// Mitsubishi GX Works2 project: 13   PLC: FX3G

// task Task_01 (event TRUE, interval 0, priority 31): POU_01

PROGRAM POU_01
VAR
  wstep : INT;
  ton1 : TON;
  ii : INT;
END_VAR
IF M8002 THEN
	wstep := 0;
END_IF;

IF NOT M0 THEN
	wstep := 0;
END_IF;

CASE wstep OF
	0:
		FOR ii := 0 TO 3 BY 1 DO
			Z0 := ii;
			Y0Z0 := FALSE;
		END_FOR;
		
		IF M0 THEN
			wstep := 20;
		END_IF;
				
	20:
		Y3 := FALSE;
		Y0 := TRUE;
		ton1(IN := TRUE, PT := T#2s);
		IF ton1.Q THEN
			ton1(IN := FALSE);
			wstep := 21;
		END_IF;
		
	21:
		Y0 := FALSE;
		Y1 := TRUE;
		ton1(IN := TRUE, PT := T#2s);
		IF ton1.Q THEN
			ton1(IN := FALSE);
			wstep := 22;
		END_IF;
		
	22:
		Y1 := FALSE;
		Y2 := TRUE;
		ton1(IN := TRUE, PT := T#3s);
		IF ton1.Q THEN
			ton1(IN := FALSE);
			wstep := 23;
		END_IF;
		
	23:
		Y2 := FALSE;
		Y3 := TRUE;
		ton1(IN := TRUE, PT := T#3s);
		IF ton1.Q THEN
			ton1(IN := FALSE);
			wstep := 0;
		END_IF;
END_CASE;
END_PROGRAM
